// Mitsubishi GX Works2 project: ZP_funtion_EX4_Addv   PLC: Q03UDV

PROGRAM MAIN
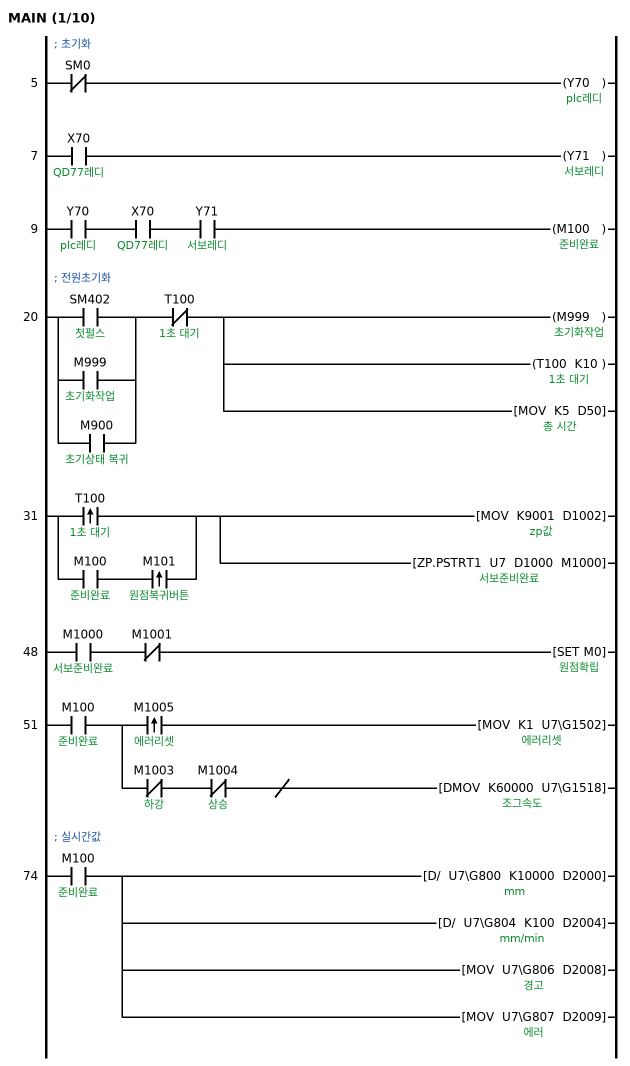
; 초기화
5     LDI     SM0
      OUT     Y70  ; plc레디
7     LD      X70  ; QD77레디
      OUT     Y71  ; 서보레디
9     LD      Y70  ; plc레디
      AND     X70  ; QD77레디
      AND     Y71  ; 서보레디
      OUT     M100  ; 준비완료
; 전원초기화
20    LD      SM402  ; 첫펄스
      OR      M999  ; 초기화작업
      OR      M900  ; 초기상태 복귀
      ANI     T100  ; 1초 대기
      OUT     M999  ; 초기화작업
      OUT     T100 K10  ; 1초 대기
      MOV     K5 D50  ; 총 시간
31    LDP     T100  ; 1초 대기
      LD      M100  ; 준비완료
      ANDP    M101  ; 원점복귀버튼
      ORB
      MOV     K9001 D1002  ; zp값
      ZP.PSTRT1 U7 D1000 M1000  ; 서보준비완료
48    LD      M1000  ; 서보준비완료
      ANI     M1001
      SET     M0  ; 원점확립
51    LD      M100  ; 준비완료
      MPS
      ANDP    M1005  ; 에러리셋
      MOV     K1 U7\G1502  ; 에러리셋
      MPP
      ANI     M1003  ; 하강
      ANI     M1004  ; 상승
      INV
      DMOV    K60000 U7\G1518  ; 조그속도
; 실시간값
74    LD      M100  ; 준비완료
      D/      U7\G800 K10000 D2000  ; mm
      D/      U7\G804 K100 D2004  ; mm/min
      MOV     U7\G806 D2008  ; 경고
      MOV     U7\G807 D2009  ; 에러
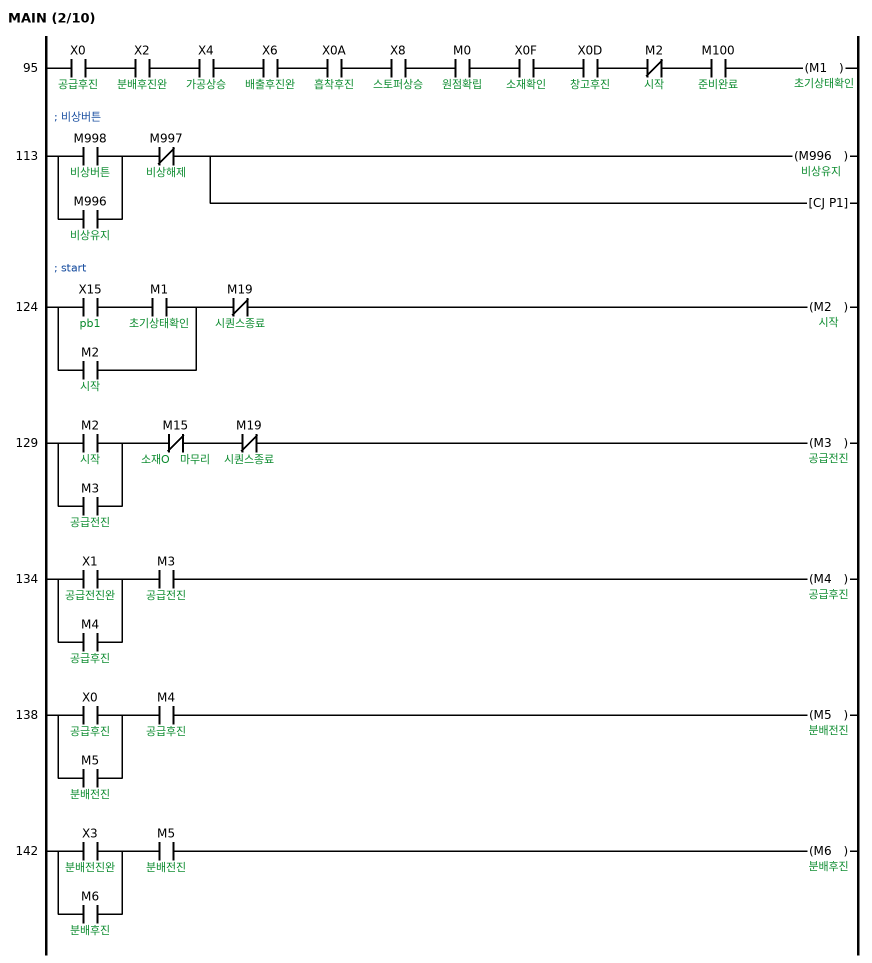
95    LD      X0  ; 공급후진
      AND     X2  ; 분배후진완
      AND     X4  ; 가공상승
      AND     X6  ; 배출후진완
      AND     X0A  ; 흡착후진
      AND     X8  ; 스토퍼상승
      AND     M0  ; 원점확립
      AND     X0F  ; 소재확인
      AND     X0D  ; 창고후진
      ANI     M2  ; 시작
      AND     M100  ; 준비완료
      OUT     M1  ; 초기상태확인
; 비상버튼
113   LD      M998  ; 비상버튼
      OR      M996  ; 비상유지
      ANI     M997  ; 비상해제
      OUT     M996  ; 비상유지
      CJ      P1
; start
124   LD      X15  ; pb1
      AND     M1  ; 초기상태확인
      OR      M2  ; 시작
      ANI     M19  ; 시퀀스종료
      OUT     M2  ; 시작
129   LD      M2  ; 시작
      OR      M3  ; 공급전진
      ANI     M15  ; 소재O   마무리
      ANI     M19  ; 시퀀스종료
      OUT     M3  ; 공급전진
134   LD      X1  ; 공급전진완
      OR      M4  ; 공급후진
      AND     M3  ; 공급전진
      OUT     M4  ; 공급후진
138   LD      X0  ; 공급후진
      OR      M5  ; 분배전진
      AND     M4  ; 공급후진
      OUT     M5  ; 분배전진
142   LD      X3  ; 분배전진완
      OR      M6  ; 분배후진
      AND     M5  ; 분배전진
      OUT     M6  ; 분배후진
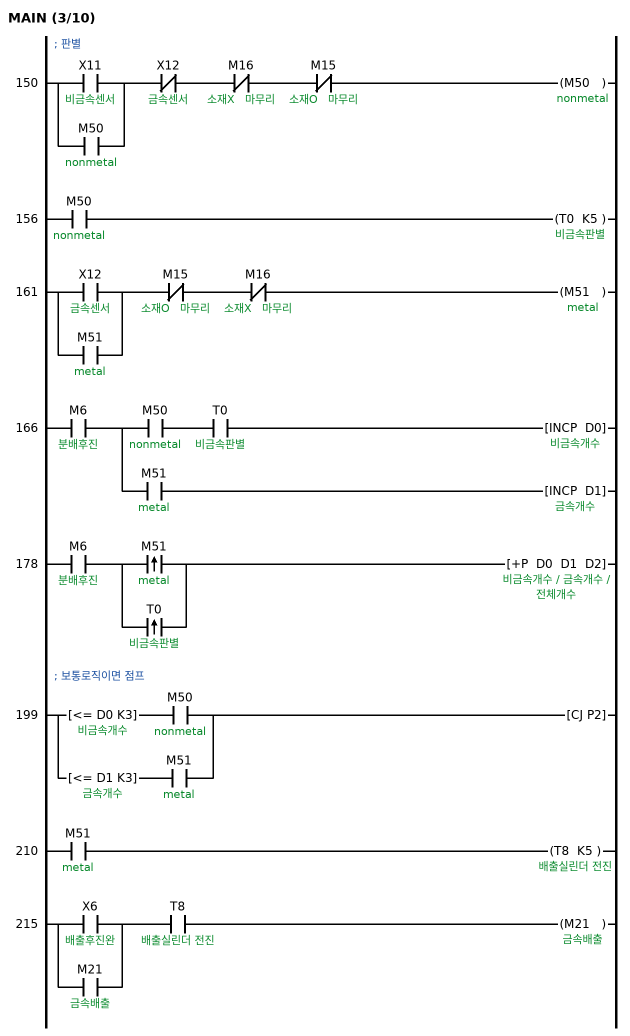
; 판별
150   LD      X11  ; 비금속센서
      OR      M50  ; nonmetal
      ANI     X12  ; 금속센서
      ANI     M16  ; 소재X   마무리
      ANI     M15  ; 소재O   마무리
      OUT     M50  ; nonmetal
156   LD      M50  ; nonmetal
      OUT     T0 K5  ; 비금속판별
161   LD      X12  ; 금속센서
      OR      M51  ; metal
      ANI     M15  ; 소재O   마무리
      ANI     M16  ; 소재X   마무리
      OUT     M51  ; metal
166   LD      M6  ; 분배후진
      MPS
      AND     M50  ; nonmetal
      AND     T0  ; 비금속판별
      INCP    D0  ; 비금속개수
      MPP
      AND     M51  ; metal
      INCP    D1  ; 금속개수
178   LD      M6  ; 분배후진
      LDP     M51  ; metal
      ORP     T0  ; 비금속판별
      ANB
      +P      D0 D1 D2  ; 전체개수
; 보통로직이면 점프
199   LD<=    D0 K3  ; 비금속개수
      AND     M50  ; nonmetal
      LD<=    D1 K3  ; 금속개수
      AND     M51  ; metal
      ORB
      CJ      P2  ; 보통 로직
210   LD      M51  ; metal
      OUT     T8 K5  ; 배출실린더 전진
215   LD      X6  ; 배출후진완
      OR      M21  ; 금속배출
      AND     T8  ; 배출실린더 전진
      OUT     M21  ; 금속배출
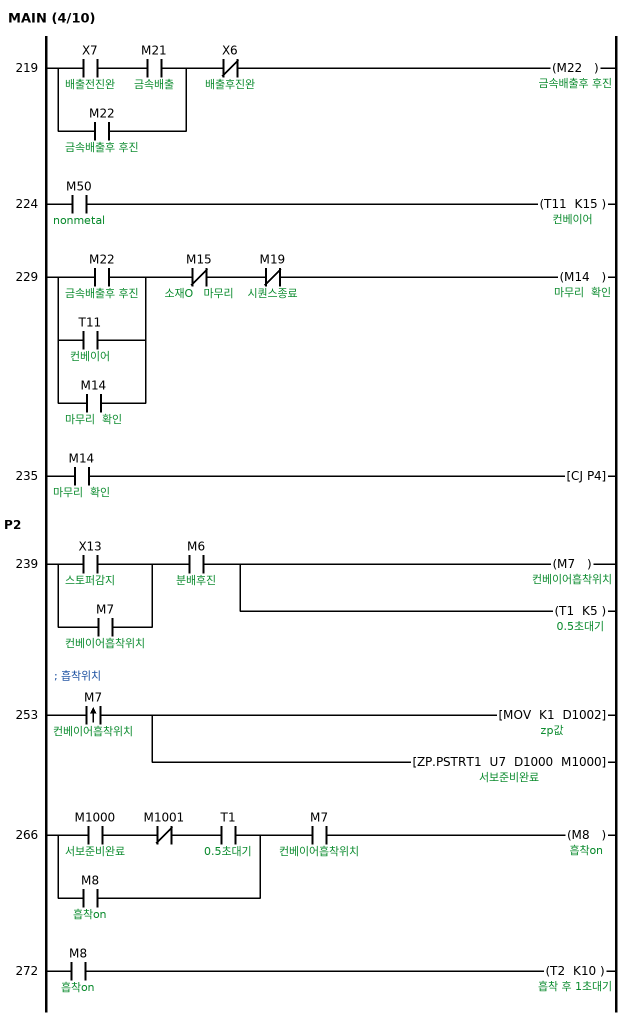
219   LD      X7  ; 배출전진완
      AND     M21  ; 금속배출
      OR      M22  ; 금속배출후 후진
      ANI     X6  ; 배출후진완
      OUT     M22  ; 금속배출후 후진
224   LD      M50  ; nonmetal
      OUT     T11 K15  ; 컨베이어
229   LD      M22  ; 금속배출후 후진
      OR      T11  ; 컨베이어
      OR      M14  ; 마무리  확인
      ANI     M15  ; 소재O   마무리
      ANI     M19  ; 시퀀스종료
      OUT     M14  ; 마무리  확인
235   LD      M14  ; 마무리  확인
      CJ      P4  ; 보통로직 다 스킵
      P2
239   LD      X13  ; 스토퍼감지
      OR      M7  ; 컨베이어흡착위치
      AND     M6  ; 분배후진
      OUT     M7  ; 컨베이어흡착위치
      OUT     T1 K5  ; 0.5초대기
; 흡착위치
253   LDP     M7  ; 컨베이어흡착위치
      MOV     K1 D1002
      ZP.PSTRT1 U7 D1000 M1000
266   LD      M1000  ; 서보준비완료
      ANI     M1001
      AND     T1  ; 0.5초대기
      OR      M8  ; 흡착on
      AND     M7  ; 컨베이어흡착위치
      OUT     M8  ; 흡착on
272   LD      M8  ; 흡착on
      OUT     T2 K10  ; 흡착 후 1초대기
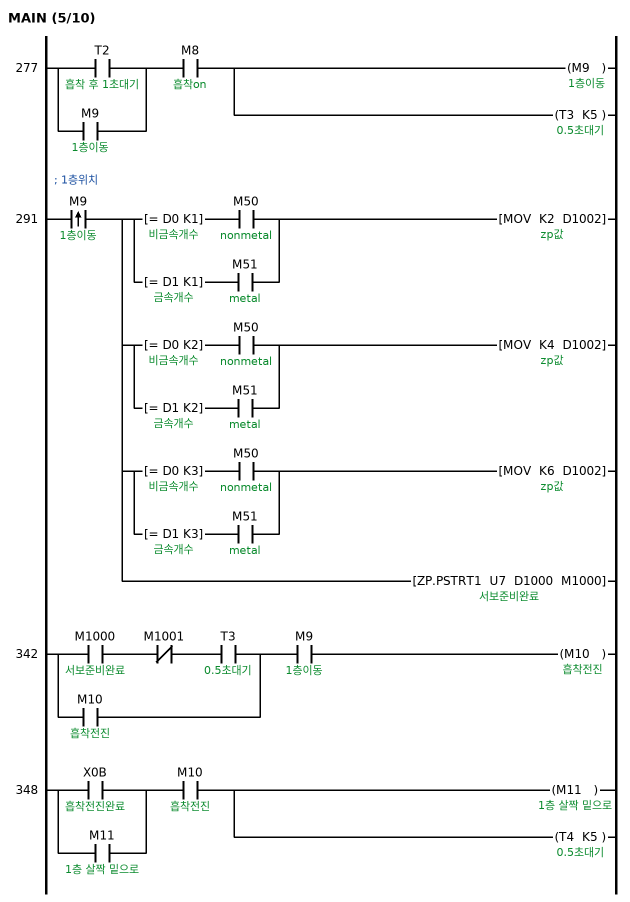
277   LD      T2  ; 흡착 후 1초대기
      OR      M9  ; 1층이동
      AND     M8  ; 흡착on
      OUT     M9  ; 1층이동
      OUT     T3 K5  ; 0.5초대기
; 1층위치
291   LDP     M9  ; 1층이동
      MPS
      LD=     D0 K1  ; 비금속개수
      AND     M50  ; nonmetal
      LD=     D1 K1  ; 금속개수
      AND     M51  ; metal
      ORB
      ANB
      MOV     K2 D1002
      MRD
      LD=     D0 K2  ; 비금속개수
      AND     M50  ; nonmetal
      LD=     D1 K2  ; 금속개수
      AND     M51  ; metal
      ORB
      ANB
      MOV     K4 D1002
      MRD
      LD=     D0 K3  ; 비금속개수
      AND     M50  ; nonmetal
      LD=     D1 K3  ; 금속개수
      AND     M51  ; metal
      ORB
      ANB
      MOV     K6 D1002
      MPP
      ZP.PSTRT1 U7 D1000 M1000
342   LD      M1000  ; 서보준비완료
      ANI     M1001
      AND     T3  ; 0.5초대기
      OR      M10  ; 흡착전진
      AND     M9  ; 1층이동
      OUT     M10  ; 흡착전진
348   LD      X0B  ; 흡착전진완료
      OR      M11  ; 1층 살짝 밑으로
      AND     M10  ; 흡착전진
      OUT     M11  ; 1층 살짝 밑으로
      OUT     T4 K5  ; 0.5초대기
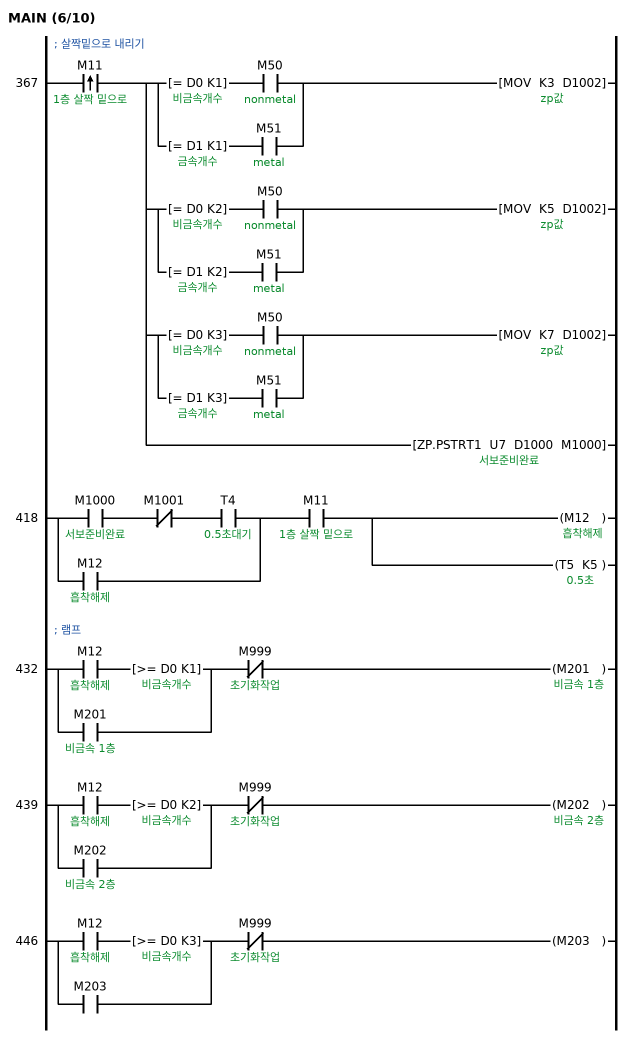
; 살짝밑으로 내리기
367   LDP     M11  ; 1층 살짝 밑으로
      MPS
      LD=     D0 K1  ; 비금속개수
      AND     M50  ; nonmetal
      LD=     D1 K1  ; 금속개수
      AND     M51  ; metal
      ORB
      ANB
      MOV     K3 D1002
      MRD
      LD=     D0 K2  ; 비금속개수
      AND     M50  ; nonmetal
      LD=     D1 K2  ; 금속개수
      AND     M51  ; metal
      ORB
      ANB
      MOV     K5 D1002
      MRD
      LD=     D0 K3  ; 비금속개수
      AND     M50  ; nonmetal
      LD=     D1 K3  ; 금속개수
      AND     M51  ; metal
      ORB
      ANB
      MOV     K7 D1002
      MPP
      ZP.PSTRT1 U7 D1000 M1000
418   LD      M1000  ; 서보준비완료
      ANI     M1001
      AND     T4  ; 0.5초대기
      OR      M12  ; 흡착해제
      AND     M11  ; 1층 살짝 밑으로
      OUT     M12  ; 흡착해제
      OUT     T5 K5  ; 0.5초
; 램프
432   LD      M12  ; 흡착해제
      AND>=   D0 K1  ; 비금속개수
      OR      M201  ; 비금속 1층
      ANI     M999  ; 초기화작업
      OUT     M201  ; 비금속 1층
439   LD      M12  ; 흡착해제
      AND>=   D0 K2  ; 비금속개수
      OR      M202  ; 비금속 2층
      ANI     M999  ; 초기화작업
      OUT     M202  ; 비금속 2층
446   LD      M12  ; 흡착해제
      AND>=   D0 K3  ; 비금속개수
      OR      M203
      ANI     M999  ; 초기화작업
      OUT     M203
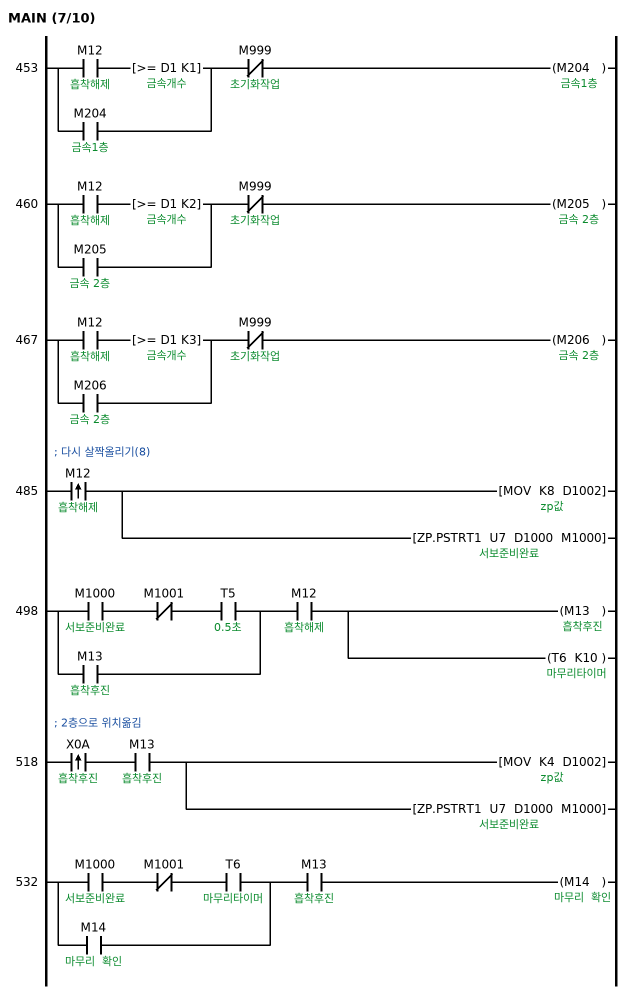
453   LD      M12  ; 흡착해제
      AND>=   D1 K1  ; 금속개수
      OR      M204  ; 금속1층
      ANI     M999  ; 초기화작업
      OUT     M204  ; 금속1층
460   LD      M12  ; 흡착해제
      AND>=   D1 K2  ; 금속개수
      OR      M205  ; 금속 2층
      ANI     M999  ; 초기화작업
      OUT     M205  ; 금속 2층
467   LD      M12  ; 흡착해제
      AND>=   D1 K3  ; 금속개수
      OR      M206  ; 금속 2층
      ANI     M999  ; 초기화작업
      OUT     M206  ; 금속 2층
; 다시 살짝올리기(8)
485   LDP     M12  ; 흡착해제
      MOV     K8 D1002
      ZP.PSTRT1 U7 D1000 M1000
498   LD      M1000  ; 서보준비완료
      ANI     M1001
      AND     T5  ; 0.5초
      OR      M13  ; 흡착후진
      AND     M12  ; 흡착해제
      OUT     M13  ; 흡착후진
      OUT     T6 K10  ; 마무리타이머
; 2층으로 위치옮김
518   LDP     X0A  ; 흡착후진
      AND     M13  ; 흡착후진
      MOV     K4 D1002
      ZP.PSTRT1 U7 D1000 M1000
532   LD      M1000  ; 서보준비완료
      ANI     M1001
      AND     T6  ; 마무리타이머
      OR      M14  ; 마무리  확인
      AND     M13  ; 흡착후진
      OUT     M14  ; 마무리  확인
      P4
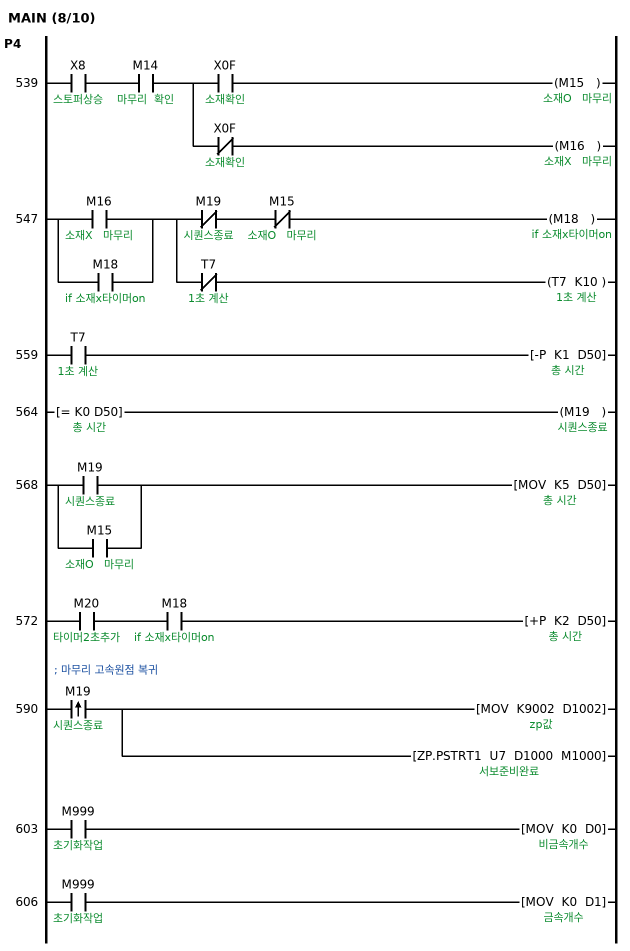
539   LD      X8  ; 스토퍼상승
      AND     M14  ; 마무리  확인
      MPS
      AND     X0F  ; 소재확인
      OUT     M15  ; 소재O   마무리
      MPP
      ANI     X0F  ; 소재확인
      OUT     M16  ; 소재X   마무리
547   LD      M16  ; 소재X   마무리
      OR      M18  ; if 소재x타이머on
      MPS
      ANI     M19  ; 시퀀스종료
      ANI     M15  ; 소재O   마무리
      OUT     M18  ; if 소재x타이머on
      MPP
      ANI     T7  ; 1초 계산
      OUT     T7 K10  ; 1초 계산
559   LD      T7  ; 1초 계산
      -P      K1 D50
564   LD=     K0 D50  ; 총 시간
      OUT     M19  ; 시퀀스종료
568   LD      M19  ; 시퀀스종료
      OR      M15  ; 소재O   마무리
      MOV     K5 D50
572   LD      M20  ; 타이머2초추가
      AND     M18  ; if 소재x타이머on
      +P      K2 D50
; 마무리 고속원점 복귀
590   LDP     M19  ; 시퀀스종료
      MOV     K9002 D1002
      ZP.PSTRT1 U7 D1000 M1000
603   LD      M999  ; 초기화작업
      MOV     K0 D0
606   LD      M999  ; 초기화작업
      MOV     K0 D1
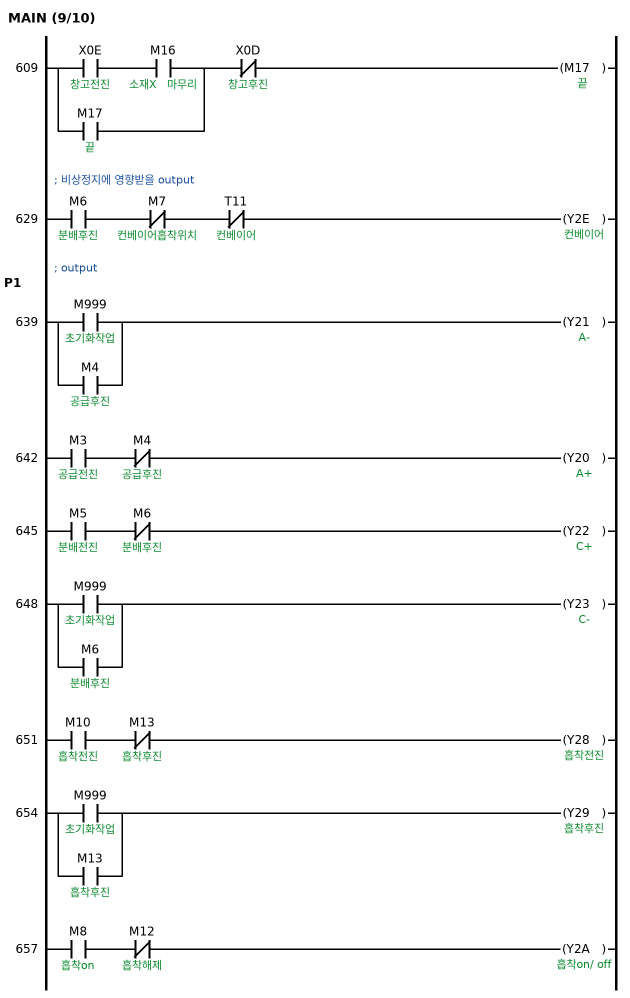
609   LD      X0E  ; 창고전진
      AND     M16  ; 소재X   마무리
      OR      M17  ; 끝
      ANI     X0D  ; 창고후진
      OUT     M17  ; 끝
; 비상정지에 영향받을 output
629   LD      M6  ; 분배후진
      ANI     M7  ; 컨베이어흡착위치
      ANI     T11  ; 컨베이어
      OUT     Y2E  ; 컨베이어
; output
      P1
639   LD      M999  ; 초기화작업
      OR      M4  ; 공급후진
      OUT     Y21  ; A-
642   LD      M3  ; 공급전진
      ANI     M4  ; 공급후진
      OUT     Y20  ; A+
645   LD      M5  ; 분배전진
      ANI     M6  ; 분배후진
      OUT     Y22  ; C+
648   LD      M999  ; 초기화작업
      OR      M6  ; 분배후진
      OUT     Y23  ; C-
651   LD      M10  ; 흡착전진
      ANI     M13  ; 흡착후진
      OUT     Y28  ; 흡착전진
654   LD      M999  ; 초기화작업
      OR      M13  ; 흡착후진
      OUT     Y29  ; 흡착후진
657   LD      M8  ; 흡착on
      ANI     M12  ; 흡착해제
      OUT     Y2A  ; 흡착on/ off
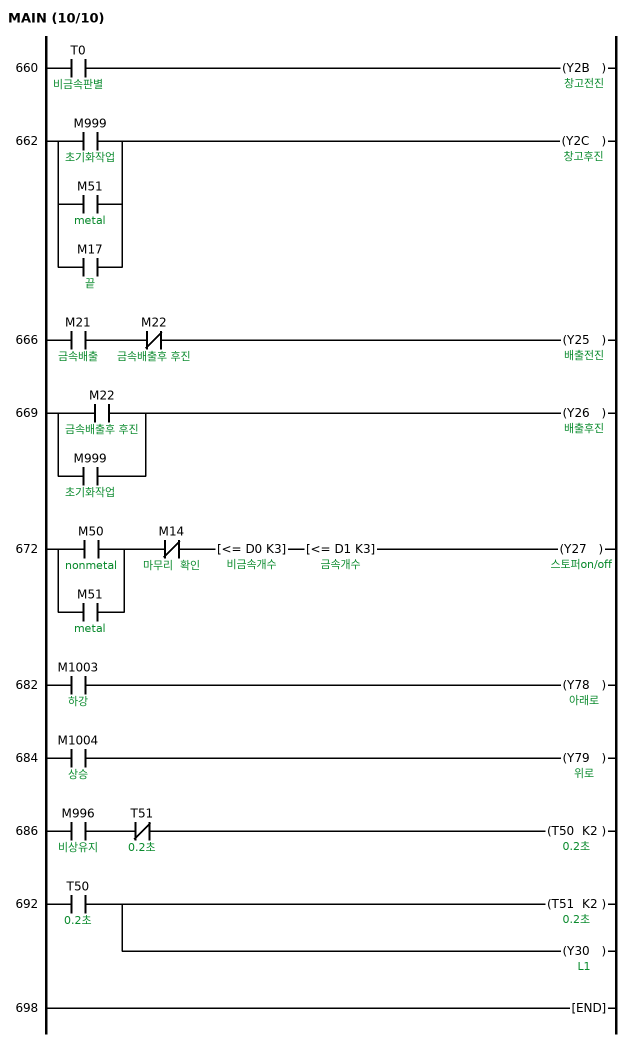
660   LD      T0  ; 비금속판별
      OUT     Y2B  ; 창고전진
662   LD      M999  ; 초기화작업
      OR      M51  ; metal
      OR      M17  ; 끝
      OUT     Y2C  ; 창고후진
666   LD      M21  ; 금속배출
      ANI     M22  ; 금속배출후 후진
      OUT     Y25  ; 배출전진
669   LD      M22  ; 금속배출후 후진
      OR      M999  ; 초기화작업
      OUT     Y26  ; 배출후진
672   LD      M50  ; nonmetal
      OR      M51  ; metal
      ANI     M14  ; 마무리  확인
      AND<=   D0 K3  ; 비금속개수
      AND<=   D1 K3  ; 금속개수
      OUT     Y27  ; 스토퍼on/off
682   LD      M1003  ; 하강
      OUT     Y78  ; 아래로
684   LD      M1004  ; 상승
      OUT     Y79  ; 위로
686   LD      M996  ; 비상유지
      ANI     T51  ; 0.2초
      OUT     T50 K2  ; 0.2초
692   LD      T50  ; 0.2초
      OUT     T51 K2  ; 0.2초
      OUT     Y30  ; L1
698   END
END_PROGRAM

// device comments not shown above
T9  ; 1초대기
T10  ; 1초대기
D5  ; 초기5초
D51  ; 몇초남았는지
P3  ; 대기동안
